FUNCTION_BLOCK FB_System_HOHW_Ablaufsteuerung
VAR_IN_OUT
	Zustand					: ST_System_HOHW_Zustand;
	Stellwert				: ST_System_HOHW_Stellwert;
	Steuerung				: ST_System_HOHW_Steuerung;
END_VAR
VAR_INPUT
	Zustand_Regelventil		: ST_RV_Zustand;
	Zustand_Pumpe			: ST_PU_Zustand;
END_VAR
VAR_OUTPUT
END_VAR
VAR
	Zustand_Stellventil: BOOL;
END_VAR

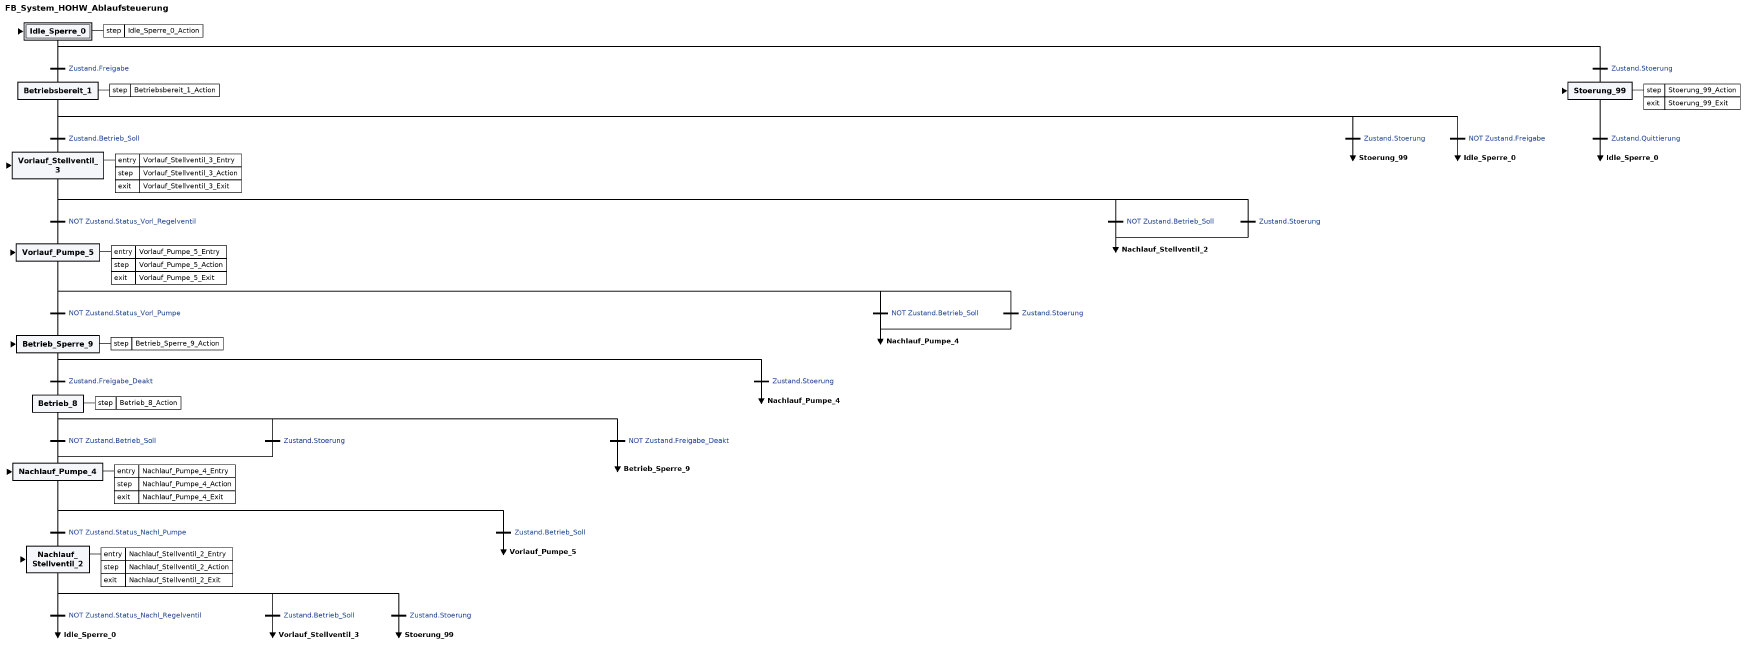
INITIAL_STEP Idle_Sperre_0:
    Idle_Sperre_0_Action(N);  // step action
END_STEP
TRANSITION FROM Idle_Sperre_0 TO Betriebsbereit_1
    := Zustand.Freigabe;
END_TRANSITION
TRANSITION FROM Idle_Sperre_0 TO Stoerung_99
    := Zustand.Stoerung;
END_TRANSITION
STEP Stoerung_99:
    Stoerung_99_Action(N);  // step action
    Stoerung_99_Exit(P0);  // exit action
END_STEP
TRANSITION FROM Stoerung_99 TO Idle_Sperre_0
    := Zustand.Quittierung;
END_TRANSITION
STEP Betriebsbereit_1:
    Betriebsbereit_1_Action(N);  // step action
END_STEP
TRANSITION FROM Betriebsbereit_1 TO Vorlauf_Stellventil_3
    := Zustand.Betrieb_Soll;
END_TRANSITION
TRANSITION FROM Betriebsbereit_1 TO Stoerung_99
    := Zustand.Stoerung;
END_TRANSITION
TRANSITION FROM Betriebsbereit_1 TO Idle_Sperre_0
    := NOT Zustand.Freigabe;
END_TRANSITION
STEP Vorlauf_Stellventil_3:
    Vorlauf_Stellventil_3_Entry(P1);  // entry action
    Vorlauf_Stellventil_3_Action(N);  // step action
    Vorlauf_Stellventil_3_Exit(P0);  // exit action
END_STEP
TRANSITION FROM Vorlauf_Stellventil_3 TO Vorlauf_Pumpe_5
    := NOT Zustand.Status_Vorl_Regelventil;
END_TRANSITION
TRANSITION FROM Vorlauf_Stellventil_3 TO Nachlauf_Stellventil_2
    := NOT Zustand.Betrieb_Soll;
END_TRANSITION
TRANSITION FROM Vorlauf_Stellventil_3 TO Nachlauf_Stellventil_2
    := Zustand.Stoerung;
END_TRANSITION
STEP Vorlauf_Pumpe_5:
    Vorlauf_Pumpe_5_Entry(P1);  // entry action
    Vorlauf_Pumpe_5_Action(N);  // step action
    Vorlauf_Pumpe_5_Exit(P0);  // exit action
END_STEP
TRANSITION FROM Vorlauf_Pumpe_5 TO Betrieb_Sperre_9
    := NOT Zustand.Status_Vorl_Pumpe;
END_TRANSITION
TRANSITION FROM Vorlauf_Pumpe_5 TO Nachlauf_Pumpe_4
    := NOT Zustand.Betrieb_Soll;
END_TRANSITION
TRANSITION FROM Vorlauf_Pumpe_5 TO Nachlauf_Pumpe_4
    := Zustand.Stoerung;
END_TRANSITION
STEP Betrieb_Sperre_9:
    Betrieb_Sperre_9_Action(N);  // step action
END_STEP
TRANSITION FROM Betrieb_Sperre_9 TO Betrieb_8
    := Zustand.Freigabe_Deakt;
END_TRANSITION
TRANSITION FROM Betrieb_Sperre_9 TO Nachlauf_Pumpe_4
    := Zustand.Stoerung;
END_TRANSITION
STEP Betrieb_8:
    Betrieb_8_Action(N);  // step action
END_STEP
TRANSITION FROM Betrieb_8 TO Nachlauf_Pumpe_4
    := NOT Zustand.Betrieb_Soll;
END_TRANSITION
TRANSITION FROM Betrieb_8 TO Nachlauf_Pumpe_4
    := Zustand.Stoerung;
END_TRANSITION
TRANSITION FROM Betrieb_8 TO Betrieb_Sperre_9
    := NOT Zustand.Freigabe_Deakt;
END_TRANSITION
STEP Nachlauf_Pumpe_4:
    Nachlauf_Pumpe_4_Entry(P1);  // entry action
    Nachlauf_Pumpe_4_Action(N);  // step action
    Nachlauf_Pumpe_4_Exit(P0);  // exit action
END_STEP
TRANSITION FROM Nachlauf_Pumpe_4 TO Nachlauf_Stellventil_2
    := NOT Zustand.Status_Nachl_Pumpe;
END_TRANSITION
TRANSITION FROM Nachlauf_Pumpe_4 TO Vorlauf_Pumpe_5
    := Zustand.Betrieb_Soll;
END_TRANSITION
STEP Nachlauf_Stellventil_2:
    Nachlauf_Stellventil_2_Entry(P1);  // entry action
    Nachlauf_Stellventil_2_Action(N);  // step action
    Nachlauf_Stellventil_2_Exit(P0);  // exit action
END_STEP
TRANSITION FROM Nachlauf_Stellventil_2 TO Idle_Sperre_0
    := NOT Zustand.Status_Nachl_Regelventil;
END_TRANSITION
TRANSITION FROM Nachlauf_Stellventil_2 TO Vorlauf_Stellventil_3
    := Zustand.Betrieb_Soll;
END_TRANSITION
TRANSITION FROM Nachlauf_Stellventil_2 TO Stoerung_99
    := Zustand.Stoerung;
END_TRANSITION

ACTION Betrieb_8_Action:
(* Stellwert setzen *)
Stellwert.Anford_Stellventil	:= TRUE;
Stellwert.Anford_Pumpe	:= TRUE;
Stellwert.Freigabe_Anlage	:= TRUE;

(* Zustand setzen *)
Zustand.Status				:= E_System_HO_Zustand_Status_Betrieb;
END_ACTION

ACTION Betrieb_Sperre_9_Action:
(* Stellwert setzen *)
Stellwert.Anford_Stellventil	:= TRUE;
Stellwert.Anford_Pumpe	:= TRUE;
Stellwert.Freigabe_Anlage	:= TRUE;

(* Zustand setzen *)
Zustand.Status				:= E_System_HO_Zustand_Status_Betrieb_Sperre;
END_ACTION

ACTION Betriebsbereit_1_Action:
(* Stellwert setzen *)
Stellwert.Anford_Stellventil	:= FALSE;
Stellwert.Anford_Pumpe	:= FALSE;
Stellwert.Freigabe_Anlage	:= FALSE;

(* Zustand setzen *)
Zustand.Status			:= E_System_HO_Zustand_Status_Betriebsbereit;
END_ACTION

ACTION Idle_Sperre_0_Action:
(* Stellwert setzen *)
Stellwert.Anford_Stellventil	:= FALSE;
Stellwert.Anford_Pumpe	:= FALSE;
Stellwert.Freigabe_Anlage	:= FALSE;

(* Zustand setzen *)
Zustand.Status			:= E_System_HO_Zustand_Status_Idle_Sperre;

(* Quittierungszustand auf False setzen, damit das System bei einer erneuten Störung nicht direkt wieder angeschaltet wird *)
Steuerung.Quittierung	:= FALSE;
END_ACTION

ACTION Nachlauf_Pumpe_4_Action:
(* Stellwert setzen *)
Stellwert.Anford_Stellventil	:= TRUE;
Stellwert.Anford_Pumpe	:= FALSE;
Stellwert.Freigabe_Anlage	:= FALSE;

(* Zustand setzen *)
Zustand.Status				:= E_System_HO_Zustand_Status_Nachl_Pumpe;
Zustand.Status_Nachl_Pumpe	:= Zustand_Pumpe.Betrieb OR Zustand_Pumpe.Status_Nachl;
END_ACTION

ACTION Nachlauf_Pumpe_4_Entry:
Zustand.Status_Nachl_Pumpe	:= TRUE;
END_ACTION

ACTION Nachlauf_Pumpe_4_Exit:
Zustand.Status_Nachl_Pumpe	:= FALSE;
END_ACTION

ACTION Nachlauf_Stellventil_2_Action:
(* Stellwert setzen *)
Stellwert.Anford_Stellventil	:= FALSE;
Stellwert.Anford_Pumpe	:= FALSE;
Stellwert.Freigabe_Anlage	:= FALSE;

(* Zustand setzen *)
Zustand.Status				:= E_System_HO_Zustand_Status_Nachl_Regelventil;
Zustand.Status_Nachl_Regelventil	:= Zustand_Regelventil.Betrieb OR Zustand_Regelventil.Status_Nachl;
END_ACTION

ACTION Nachlauf_Stellventil_2_Entry:
Zustand.Status_Nachl_Regelventil	:= TRUE;
END_ACTION

ACTION Nachlauf_Stellventil_2_Exit:
Zustand.Status_Nachl_Regelventil	:= FALSE;
END_ACTION

ACTION Stoerung_99_Action:
(* Stellwert setzen *)
Stellwert.Anford_Stellventil	:= FALSE;
Stellwert.Anford_Pumpe	:= FALSE;
Stellwert.Freigabe_Anlage	:= FALSE;

(* Zustand setzen *)
Zustand.Stoerung			:= TRUE;
Zustand.Status			:= E_System_HO_Zustand_Status_Stoerung;
END_ACTION

ACTION Stoerung_99_Exit:
Zustand.Stoerung	:= FALSE;
END_ACTION

ACTION Vorlauf_Pumpe_5_Action:
(* Stellwert setzen *)
Stellwert.Anford_Stellventil	:= TRUE;
Stellwert.Anford_Pumpe	:= TRUE;
Stellwert.Freigabe_Anlage	:= FALSE;

(* Zustand setzen *)
Zustand.Status				:= E_System_HO_Zustand_Status_Vorl_Pumpe;
Zustand.Status_Vorl_Pumpe	:= NOT(Zustand_Pumpe.Betrieb AND NOT Zustand_Pumpe.Status_Vorl);
END_ACTION

ACTION Vorlauf_Pumpe_5_Entry:
Zustand.Status_Vorl_Pumpe	:= TRUE;
END_ACTION

ACTION Vorlauf_Pumpe_5_Exit:
Zustand.Status_Vorl_Pumpe	:= FALSE;
END_ACTION

ACTION Vorlauf_Stellventil_3_Action:
(* Stellwert setzen *)
Stellwert.Anford_Stellventil	:= TRUE;
Stellwert.Anford_Pumpe	:= FALSE;
Stellwert.Freigabe_Anlage	:= FALSE;

(* Zustand setzen *)
Zustand.Status				:= E_System_HO_Zustand_Status_Vorl_Regelventil;
Zustand.Status_Vorl_Regelventil	:= NOT(Zustand_Regelventil.Betrieb AND NOT Zustand_Regelventil.Status_Vorl);
END_ACTION

ACTION Vorlauf_Stellventil_3_Entry:
Zustand.Status_Vorl_Regelventil	:= TRUE;
END_ACTION

ACTION Vorlauf_Stellventil_3_Exit:
Zustand.Status_Vorl_Regelventil	:= FALSE;
END_ACTION

END_FUNCTION_BLOCK

(* stored: Version 1.1.0.1, ProductVersion 3.1.4024.9
   POU FB_System_HOHW_Ablaufsteuerung: Id {c6c69ed0-091f-4721-a6cb-766c62bad267}, SpecialFunc None
   Action Betrieb_8_Action: Id {0a697c78-afed-482f-8628-a69b6d71bd25}
   Action Betrieb_Sperre_9_Action: Id {b7c521da-35b9-4ac8-9d20-cafc54a3ca59}
   Action Betriebsbereit_1_Action: Id {34a0fb91-35af-481a-900b-3db6e7a8625b}
   Action Idle_Sperre_0_Action: Id {7c751a14-c4e3-4400-bd15-993acd299bb3}
   Action Nachlauf_Pumpe_4_Action: Id {710dd306-8846-4b23-a5b3-26be276211c6}
   Action Nachlauf_Pumpe_4_Entry: Id {92aab707-8f99-4149-b2a1-8fb42d01333d}
   Action Nachlauf_Pumpe_4_Exit: Id {1702cd00-fc04-45d8-a43b-5056386f696a}
   Action Nachlauf_Stellventil_2_Action: Id {e66c597e-4803-4267-aa6d-7386331df9cd}
   Action Nachlauf_Stellventil_2_Entry: Id {590cfcdb-ea6c-4dd3-80a7-0f59eba5f2b0}
   Action Nachlauf_Stellventil_2_Exit: Id {95a5d83e-fc9f-4404-ad24-e64337b83457}
   Action Stoerung_99_Action: Id {c8421be7-a66f-4af5-a980-491a4028f97e}
   Action Stoerung_99_Exit: Id {1fd0d7e0-7999-4163-b407-de138b92eb22}
   Action Vorlauf_Pumpe_5_Action: Id {2a402a37-b755-4df3-9746-fa416780d7ce}
   Action Vorlauf_Pumpe_5_Entry: Id {a7b74c65-b2ba-40a2-837f-9b51c887f3cf}
   Action Vorlauf_Pumpe_5_Exit: Id {7986cab6-ce56-4e49-aa90-b508c14fb4f2}
   Action Vorlauf_Stellventil_3_Action: Id {6d63eef1-4f82-4d34-994a-b6925c787cae}
   Action Vorlauf_Stellventil_3_Entry: Id {50d7f56b-f127-46b9-b5ba-d2c3e9bc57d4}
   Action Vorlauf_Stellventil_3_Exit: Id {bd1e9cc8-3dd3-451f-a3ec-1b7379d7e0df} *)
